INTERFACE PUBLIC CompletingCommands EXTENDS RunningStateCommands, ActionStateCommands

END_INTERFACE

(* stored: Version 1.1.0.1, ProductVersion 3.1.4026.18
   Itf CompletingCommands: Id {81f78d50-be70-0fcb-055f-f4ffcddca7b0} *)
